FUNCTION_BLOCK ENCODER_AXIS_SINGLE_PHASE (* Composite Function Block Type *)
  (* Standard: 61499-2 *)
  (* Version 0.0, 1/25/2023, Dmitrii, Flexbridge AB, template *)
  PACKAGE UAO.Hackathon;
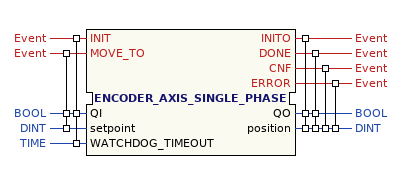
  EVENT_INPUT
    INIT WITH QI, WATCHDOG_TIMEOUT; (* Initialization Request *)
    MOVE_TO WITH QI, setpoint; (* Trigger movement to the setpoint *)
  END_EVENT
  EVENT_OUTPUT
    INITO WITH QO, position; (* Initialization Confirm *)
    DONE WITH QO, position; (* Execution Confirmation *)
    CNF WITH position; (* Position update confirmation *)
    ERROR WITH position; (* Error: stopped by timeout *)
  END_EVENT
  VAR_INPUT
    QI : BOOL; (* Input event qualifier *)
    setpoint : DINT;
    WATCHDOG_TIMEOUT : TIME; (* Delay Time *)
  END_VAR
  VAR_OUTPUT
    QO : BOOL; (* Output event qualifier *)
    position : DINT;
  END_VAR
  FBS
    watchdog : E_DELAY;
    MotorDriver : MOTOR_DRIVER_SIMPLE;
    FineMove : STEPPER;
    StepTimeout : E_DELAY(DT := T#10ms);
    BackwardFlag : COMPARE_112C76C471B7A99C2; {SET_ATTRIBUTE(Configuration.GenericFBType.InterfaceParams, Runtime.Standard#CNT:=2;IN${CNT$}:DINT)}
    SensorDriver : SENSOR_DRIVER_SINGLE_PHASE;
    InitMoveHome : SIMPLE_INIT;
    WaitPositionUpdate : E_DELAY(DT := T#200ms);
    Position : POSITION_MONITOR_V2;
    CoarseMove : COARSE_MOVE_V2(threshold := 30);
    RefSwitchDelay : E_DELAY(DT := T#50ms);
    DelayPositionReset : E_DELAY(DT := T#100ms);
  END_FBS
  EVENT_CONNECTIONS
    FineMove.START_STEP_TIMEOUT TO StepTimeout.START;
    StepTimeout.EO TO FineMove.STEP_TIMEOUT;
    FineMove.MOVE_FORWARD TO MotorDriver.MOVE_FORWARD;
    FineMove.MOVE_BACKWARD TO MotorDriver.MOVE_BACKWARD;
    FineMove.STOP TO MotorDriver.STOP;
    FineMove.DONE TO DONE;
    MOVE_TO TO BackwardFlag.REQ;
    MOVE_TO TO watchdog.START;
    FineMove.DONE TO watchdog.STOP;
    watchdog.EO TO MotorDriver.STOP;
    INIT TO SensorDriver.INIT;
    SensorDriver.INITO TO MotorDriver.INIT;
    RefSwitchDelay.EO TO MotorDriver.STOP;
    RefSwitchDelay.EO TO Position.RESET;
    MotorDriver.INITO TO InitMoveHome.INIT;
    InitMoveHome.INITO TO INITO;
    SensorDriver.CNF TO InitMoveHome.REQ;
    watchdog.EO TO InitMoveHome.ERROR;
    InitMoveHome.MOTOR_ON TO MotorDriver.MOVE_BACKWARD;
    InitMoveHome.MOTOR_OFF TO MotorDriver.STOP;
    BackwardFlag.CNF TO CoarseMove.TRIGGER;
    RefSwitchDelay.EO TO CoarseMove.HOME;
    Position.CNF TO CoarseMove.REQ;
    CoarseMove.MOVE_FORWARD TO MotorDriver.MOVE_FORWARD;
    CoarseMove.MOVE_BACKWARD TO MotorDriver.MOVE_BACKWARD;
    CoarseMove.STOP TO MotorDriver.STOP;
    InitMoveHome.INITO TO SensorDriver.HSC_START;
    CoarseMove.DONE TO WaitPositionUpdate.START;
    WaitPositionUpdate.EO TO FineMove.TRIGGER;
    Position.CNF TO CNF;
    Position.RESET_COUNTER TO SensorDriver.HSC_SYNC;
    SensorDriver.CNF TO Position.CNT_UPDATE;
    CoarseMove.STOP TO Position.STOP_IND;
    FineMove.STOP TO Position.STOP_IND;
    SensorDriver.RefSwitch_EO TO RefSwitchDelay.START;
    InitMoveHome.INITO TO Position.RESET;
    Position.CAPTUREO TO FineMove.REQ;
    watchdog.EO TO ERROR;
    watchdog.EO TO Position.STOP_IND;
    CoarseMove.FORCE_RESET TO DelayPositionReset.START;
    DelayPositionReset.EO TO Position.RESET;
    SensorDriver.CNF TO CoarseMove.REQ;
  END_CONNECTIONS
  DATA_CONNECTIONS
    WATCHDOG_TIMEOUT TO watchdog.DT;
    setpoint TO FineMove.setpoint;
    setpoint TO BackwardFlag.IN1;
    BackwardFlag.LT TO Position.backwardFlag;
    BackwardFlag.LT TO FineMove.backwardFlag;
    QI TO SensorDriver.QI;
    SensorDriver.QO TO MotorDriver.QI;
    InitMoveHome.QO TO QO;
    MotorDriver.QO TO InitMoveHome.QI;
    SensorDriver.switch TO InitMoveHome.switch;
    setpoint TO CoarseMove.setpoint;
    SensorDriver.counter TO Position.counter;
    Position.position TO FineMove.position;
    Position.position TO CoarseMove.position;
    Position.position TO position;
    Position.capturedPosition TO BackwardFlag.IN2;
    SensorDriver.switch TO CoarseMove.refSwitch;
  END_CONNECTIONS
END_FUNCTION_BLOCK
